DATA_BLOCK "RSE_GLOBAL_DB"
TITLE = Report System Error Diagnostic Block
{ S7_Optimized_Access := 'FALSE' }
AUTHOR : SIMATIC
FAMILY : RSEDIAG
NAME : RSE
VERSION : 1.0
NON_RETAIN
// This DB contains the generated data from STEP 7 Report System Errors.
   STRUCT
      DB_Nummer { ExternalVisible := 'False'} : Word;
      DB_Init { ExternalVisible := 'False'} : Bool;
      HotRestart { ExternalVisible := 'False'} : Bool;
      DB_bZaehler { ExternalVisible := 'False'} : Byte;
      TraceZyklusNo { ExternalVisible := 'False'} : Word;
      TraceZyklusAuswertung { ExternalVisible := 'False'} : Word;
      TraceZyklus126No { ExternalVisible := 'False'} : Word;
      TraceZyklus127No { ExternalVisible := 'False'} : Word;
      TraceStatus1 { ExternalVisible := 'False'} : Word;
      TraceMeldungenAnzahl { ExternalVisible := 'False'} : Byte;
      TraceMeldungenMax { ExternalVisible := 'False'} : Byte;
      Daten { ExternalVisible := 'False'} : Array[1..805] of Byte;
      DiagSZLHeader { ExternalVisible := 'False'} : Struct
         LENTHDR { ExternalVisible := 'False'} : Word;
         N_DR { ExternalVisible := 'False'} : Word;
      END_STRUCT;
      SZLHeader { ExternalVisible := 'False'} : Struct
         LENTHDR { ExternalVisible := 'False'} : Word;
         N_DR { ExternalVisible := 'False'} : Word;
      END_STRUCT;
   END_STRUCT;


BEGIN
   DB_Nummer := WORD#16#0032;
   Daten[1] := BYTE#16#08;
   Daten[4] := BYTE#16#09;
   Daten[5] := BYTE#16#03;
   Daten[6] := BYTE#16#58;
   Daten[7] := BYTE#16#03;
   Daten[8] := BYTE#16#26;
   Daten[9] := BYTE#16#03;
   Daten[10] := BYTE#16#28;
   Daten[11] := BYTE#16#03;
   Daten[12] := BYTE#16#2A;
   Daten[13] := BYTE#16#03;
   Daten[14] := BYTE#16#2C;
   Daten[15] := BYTE#16#03;
   Daten[16] := BYTE#16#2E;
   Daten[17] := BYTE#16#03;
   Daten[18] := BYTE#16#30;
   Daten[19] := BYTE#16#03;
   Daten[20] := BYTE#16#56;
   Daten[21] := BYTE#16#03;
   Daten[22] := BYTE#16#3C;
   Daten[23] := BYTE#16#01;
   Daten[29] := BYTE#16#08;
   Daten[30] := BYTE#16#40;
   Daten[32] := BYTE#16#04;
   Daten[33] := BYTE#16#03;
   Daten[34] := BYTE#16#66;
   Daten[35] := BYTE#16#03;
   Daten[36] := BYTE#16#46;
   Daten[37] := BYTE#16#03;
   Daten[38] := BYTE#16#44;
   Daten[39] := BYTE#16#03;
   Daten[40] := BYTE#16#42;
   Daten[51] := BYTE#16#FF;
   Daten[52] := BYTE#16#FF;
   Daten[53] := BYTE#16#FF;
   Daten[54] := BYTE#16#FF;
   Daten[56] := BYTE#16#40;
   Daten[67] := BYTE#16#FF;
   Daten[68] := BYTE#16#FF;
   Daten[69] := BYTE#16#FF;
   Daten[70] := BYTE#16#FF;
   Daten[71] := BYTE#16#03;
   Daten[72] := BYTE#16#48;
   Daten[75] := BYTE#16#04;
   Daten[79] := BYTE#16#08;
   Daten[80] := BYTE#16#08;
   Daten[85] := BYTE#16#FF;
   Daten[86] := BYTE#16#FF;
   Daten[87] := BYTE#16#FF;
   Daten[88] := BYTE#16#FF;
   Daten[93] := BYTE#16#05;
   Daten[95] := BYTE#16#06;
   Daten[99] := BYTE#16#20;
   Daten[100] := BYTE#16#04;
   Daten[109] := BYTE#16#01;
   Daten[110] := BYTE#16#FF;
   Daten[111] := BYTE#16#FF;
   Daten[112] := BYTE#16#FF;
   Daten[113] := BYTE#16#FF;
   Daten[114] := BYTE#16#07;
   Daten[116] := BYTE#16#08;
   Daten[118] := BYTE#16#05;
   Daten[120] := BYTE#16#06;
   Daten[123] := BYTE#16#20;
   Daten[124] := BYTE#16#04;
   Daten[133] := BYTE#16#01;
   Daten[134] := BYTE#16#FF;
   Daten[135] := BYTE#16#FF;
   Daten[136] := BYTE#16#FF;
   Daten[137] := BYTE#16#FF;
   Daten[138] := BYTE#16#07;
   Daten[140] := BYTE#16#08;
   Daten[142] := BYTE#16#05;
   Daten[144] := BYTE#16#06;
   Daten[147] := BYTE#16#20;
   Daten[148] := BYTE#16#04;
   Daten[152] := BYTE#16#08;
   Daten[153] := BYTE#16#08;
   Daten[157] := BYTE#16#FF;
   Daten[158] := BYTE#16#FF;
   Daten[159] := BYTE#16#FF;
   Daten[160] := BYTE#16#FF;
   Daten[161] := BYTE#16#FF;
   Daten[162] := BYTE#16#09;
   Daten[166] := BYTE#16#08;
   Daten[168] := BYTE#16#20;
   Daten[169] := BYTE#16#04;
   Daten[173] := BYTE#16#08;
   Daten[174] := BYTE#16#08;
   Daten[178] := BYTE#16#FF;
   Daten[179] := BYTE#16#FF;
   Daten[180] := BYTE#16#FF;
   Daten[181] := BYTE#16#FF;
   Daten[182] := BYTE#16#FF;
   Daten[183] := BYTE#16#09;
   Daten[187] := BYTE#16#08;
   Daten[189] := BYTE#16#20;
   Daten[190] := BYTE#16#04;
   Daten[194] := BYTE#16#08;
   Daten[195] := BYTE#16#08;
   Daten[199] := BYTE#16#FF;
   Daten[200] := BYTE#16#FF;
   Daten[201] := BYTE#16#FF;
   Daten[202] := BYTE#16#FF;
   Daten[203] := BYTE#16#FF;
   Daten[204] := BYTE#16#09;
   Daten[208] := BYTE#16#08;
   Daten[210] := BYTE#16#20;
   Daten[211] := BYTE#16#04;
   Daten[215] := BYTE#16#08;
   Daten[216] := BYTE#16#08;
   Daten[220] := BYTE#16#FF;
   Daten[221] := BYTE#16#FF;
   Daten[222] := BYTE#16#FF;
   Daten[223] := BYTE#16#FF;
   Daten[224] := BYTE#16#FF;
   Daten[225] := BYTE#16#09;
   Daten[229] := BYTE#16#08;
   Daten[231] := BYTE#16#20;
   Daten[232] := BYTE#16#04;
   Daten[236] := BYTE#16#08;
   Daten[237] := BYTE#16#08;
   Daten[241] := BYTE#16#FF;
   Daten[242] := BYTE#16#FF;
   Daten[243] := BYTE#16#FF;
   Daten[244] := BYTE#16#FF;
   Daten[245] := BYTE#16#FF;
   Daten[246] := BYTE#16#09;
   Daten[250] := BYTE#16#08;
   Daten[253] := BYTE#16#04;
   Daten[257] := BYTE#16#08;
   Daten[258] := BYTE#16#08;
   Daten[263] := BYTE#16#FF;
   Daten[264] := BYTE#16#FF;
   Daten[265] := BYTE#16#FF;
   Daten[266] := BYTE#16#FF;
   Daten[273] := BYTE#16#40;
   Daten[284] := BYTE#16#FF;
   Daten[285] := BYTE#16#FF;
   Daten[286] := BYTE#16#FF;
   Daten[287] := BYTE#16#FF;
   Daten[288] := BYTE#16#03;
   Daten[289] := BYTE#16#5C;
   Daten[292] := BYTE#16#04;
   Daten[296] := BYTE#16#08;
   Daten[297] := BYTE#16#08;
   Daten[302] := BYTE#16#FF;
   Daten[303] := BYTE#16#FF;
   Daten[304] := BYTE#16#FF;
   Daten[305] := BYTE#16#FF;
   Daten[311] := BYTE#16#08;
   Daten[312] := BYTE#16#48;
   Daten[314] := BYTE#16#04;
   Daten[315] := BYTE#16#03;
   Daten[316] := BYTE#16#3E;
   Daten[317] := BYTE#16#03;
   Daten[318] := BYTE#16#18;
   Daten[319] := BYTE#16#03;
   Daten[320] := BYTE#16#1A;
   Daten[321] := BYTE#16#03;
   Daten[322] := BYTE#16#4A;
   Daten[323] := BYTE#16#01;
   Daten[329] := BYTE#16#02;
   Daten[332] := BYTE#16#40;
   Daten[343] := BYTE#16#FF;
   Daten[344] := BYTE#16#FF;
   Daten[345] := BYTE#16#FF;
   Daten[346] := BYTE#16#FF;
   Daten[348] := BYTE#16#20;
   Daten[349] := BYTE#16#04;
   Daten[353] := BYTE#16#08;
   Daten[354] := BYTE#16#08;
   Daten[355] := BYTE#16#FF;
   Daten[356] := BYTE#16#FF;
   Daten[357] := BYTE#16#FF;
   Daten[358] := BYTE#16#FF;
   Daten[359] := BYTE#16#FF;
   Daten[360] := BYTE#16#FF;
   Daten[361] := BYTE#16#FF;
   Daten[362] := BYTE#16#FF;
   Daten[363] := BYTE#16#09;
   Daten[367] := BYTE#16#20;
   Daten[369] := BYTE#16#20;
   Daten[370] := BYTE#16#04;
   Daten[374] := BYTE#16#08;
   Daten[375] := BYTE#16#08;
   Daten[376] := BYTE#16#FF;
   Daten[377] := BYTE#16#FF;
   Daten[378] := BYTE#16#FF;
   Daten[379] := BYTE#16#FF;
   Daten[380] := BYTE#16#FF;
   Daten[381] := BYTE#16#FF;
   Daten[382] := BYTE#16#FF;
   Daten[383] := BYTE#16#FF;
   Daten[384] := BYTE#16#09;
   Daten[388] := BYTE#16#20;
   Daten[390] := BYTE#16#20;
   Daten[391] := BYTE#16#04;
   Daten[395] := BYTE#16#08;
   Daten[396] := BYTE#16#08;
   Daten[400] := BYTE#16#FF;
   Daten[401] := BYTE#16#FF;
   Daten[402] := BYTE#16#FF;
   Daten[403] := BYTE#16#FF;
   Daten[404] := BYTE#16#FF;
   Daten[405] := BYTE#16#09;
   Daten[409] := BYTE#16#08;
   Daten[410] := BYTE#16#08;
   Daten[411] := BYTE#16#48;
   Daten[413] := BYTE#16#03;
   Daten[414] := BYTE#16#03;
   Daten[415] := BYTE#16#64;
   Daten[416] := BYTE#16#03;
   Daten[417] := BYTE#16#22;
   Daten[418] := BYTE#16#03;
   Daten[419] := BYTE#16#54;
   Daten[420] := BYTE#16#01;
   Daten[426] := BYTE#16#02;
   Daten[429] := BYTE#16#40;
   Daten[440] := BYTE#16#FF;
   Daten[441] := BYTE#16#FF;
   Daten[442] := BYTE#16#FF;
   Daten[443] := BYTE#16#FF;
   Daten[446] := BYTE#16#04;
   Daten[450] := BYTE#16#08;
   Daten[451] := BYTE#16#08;
   Daten[456] := BYTE#16#FF;
   Daten[457] := BYTE#16#FF;
   Daten[458] := BYTE#16#FF;
   Daten[459] := BYTE#16#FF;
   Daten[460] := BYTE#16#09;
   Daten[465] := BYTE#16#04;
   Daten[469] := BYTE#16#08;
   Daten[470] := BYTE#16#08;
   Daten[475] := BYTE#16#FF;
   Daten[476] := BYTE#16#FF;
   Daten[477] := BYTE#16#FF;
   Daten[478] := BYTE#16#FF;
   Daten[479] := BYTE#16#09;
   Daten[482] := BYTE#16#08;
   Daten[483] := BYTE#16#48;
   Daten[485] := BYTE#16#03;
   Daten[486] := BYTE#16#03;
   Daten[487] := BYTE#16#62;
   Daten[488] := BYTE#16#03;
   Daten[489] := BYTE#16#1C;
   Daten[490] := BYTE#16#03;
   Daten[491] := BYTE#16#4C;
   Daten[492] := BYTE#16#01;
   Daten[498] := BYTE#16#02;
   Daten[501] := BYTE#16#40;
   Daten[512] := BYTE#16#FF;
   Daten[513] := BYTE#16#FF;
   Daten[514] := BYTE#16#FF;
   Daten[515] := BYTE#16#FF;
   Daten[518] := BYTE#16#04;
   Daten[522] := BYTE#16#08;
   Daten[523] := BYTE#16#08;
   Daten[528] := BYTE#16#FF;
   Daten[529] := BYTE#16#FF;
   Daten[530] := BYTE#16#FF;
   Daten[531] := BYTE#16#FF;
   Daten[532] := BYTE#16#09;
   Daten[537] := BYTE#16#04;
   Daten[541] := BYTE#16#08;
   Daten[542] := BYTE#16#08;
   Daten[547] := BYTE#16#FF;
   Daten[548] := BYTE#16#FF;
   Daten[549] := BYTE#16#FF;
   Daten[550] := BYTE#16#FF;
   Daten[551] := BYTE#16#09;
   Daten[554] := BYTE#16#08;
   Daten[555] := BYTE#16#48;
   Daten[557] := BYTE#16#03;
   Daten[558] := BYTE#16#03;
   Daten[559] := BYTE#16#5E;
   Daten[560] := BYTE#16#03;
   Daten[561] := BYTE#16#1E;
   Daten[562] := BYTE#16#03;
   Daten[563] := BYTE#16#4E;
   Daten[564] := BYTE#16#01;
   Daten[570] := BYTE#16#02;
   Daten[573] := BYTE#16#40;
   Daten[584] := BYTE#16#FF;
   Daten[585] := BYTE#16#FF;
   Daten[586] := BYTE#16#FF;
   Daten[587] := BYTE#16#FF;
   Daten[590] := BYTE#16#04;
   Daten[594] := BYTE#16#08;
   Daten[595] := BYTE#16#08;
   Daten[600] := BYTE#16#FF;
   Daten[601] := BYTE#16#FF;
   Daten[602] := BYTE#16#FF;
   Daten[603] := BYTE#16#FF;
   Daten[604] := BYTE#16#09;
   Daten[609] := BYTE#16#04;
   Daten[613] := BYTE#16#08;
   Daten[614] := BYTE#16#08;
   Daten[619] := BYTE#16#FF;
   Daten[620] := BYTE#16#FF;
   Daten[621] := BYTE#16#FF;
   Daten[622] := BYTE#16#FF;
   Daten[623] := BYTE#16#09;
   Daten[626] := BYTE#16#08;
   Daten[627] := BYTE#16#48;
   Daten[629] := BYTE#16#03;
   Daten[630] := BYTE#16#03;
   Daten[631] := BYTE#16#60;
   Daten[632] := BYTE#16#03;
   Daten[633] := BYTE#16#20;
   Daten[634] := BYTE#16#03;
   Daten[635] := BYTE#16#52;
   Daten[636] := BYTE#16#01;
   Daten[642] := BYTE#16#02;
   Daten[645] := BYTE#16#40;
   Daten[656] := BYTE#16#FF;
   Daten[657] := BYTE#16#FF;
   Daten[658] := BYTE#16#FF;
   Daten[659] := BYTE#16#FF;
   Daten[662] := BYTE#16#04;
   Daten[666] := BYTE#16#08;
   Daten[667] := BYTE#16#08;
   Daten[672] := BYTE#16#FF;
   Daten[673] := BYTE#16#FF;
   Daten[674] := BYTE#16#FF;
   Daten[675] := BYTE#16#FF;
   Daten[676] := BYTE#16#09;
   Daten[681] := BYTE#16#04;
   Daten[685] := BYTE#16#08;
   Daten[686] := BYTE#16#08;
   Daten[691] := BYTE#16#FF;
   Daten[692] := BYTE#16#FF;
   Daten[693] := BYTE#16#FF;
   Daten[694] := BYTE#16#FF;
   Daten[695] := BYTE#16#09;
   Daten[698] := BYTE#16#08;
   Daten[699] := BYTE#16#48;
   Daten[701] := BYTE#16#03;
   Daten[702] := BYTE#16#03;
   Daten[703] := BYTE#16#5A;
   Daten[704] := BYTE#16#03;
   Daten[705] := BYTE#16#24;
   Daten[706] := BYTE#16#03;
   Daten[707] := BYTE#16#50;
   Daten[708] := BYTE#16#01;
   Daten[714] := BYTE#16#02;
   Daten[717] := BYTE#16#40;
   Daten[728] := BYTE#16#FF;
   Daten[729] := BYTE#16#FF;
   Daten[730] := BYTE#16#FF;
   Daten[731] := BYTE#16#FF;
   Daten[734] := BYTE#16#04;
   Daten[738] := BYTE#16#08;
   Daten[739] := BYTE#16#08;
   Daten[744] := BYTE#16#FF;
   Daten[745] := BYTE#16#FF;
   Daten[746] := BYTE#16#FF;
   Daten[747] := BYTE#16#FF;
   Daten[748] := BYTE#16#09;
   Daten[753] := BYTE#16#04;
   Daten[757] := BYTE#16#08;
   Daten[758] := BYTE#16#08;
   Daten[763] := BYTE#16#FF;
   Daten[764] := BYTE#16#FF;
   Daten[765] := BYTE#16#FF;
   Daten[766] := BYTE#16#FF;
   Daten[767] := BYTE#16#09;
   Daten[770] := BYTE#16#08;
   Daten[771] := BYTE#16#08;
   Daten[773] := BYTE#16#06;
   Daten[774] := BYTE#16#03;
   Daten[775] := BYTE#16#40;
   Daten[776] := BYTE#16#03;
   Daten[777] := BYTE#16#34;
   Daten[778] := BYTE#16#03;
   Daten[779] := BYTE#16#36;
   Daten[780] := BYTE#16#03;
   Daten[781] := BYTE#16#38;
   Daten[782] := BYTE#16#03;
   Daten[783] := BYTE#16#32;
   Daten[784] := BYTE#16#03;
   Daten[785] := BYTE#16#3A;
   Daten[786] := BYTE#16#03;
   Daten[792] := BYTE#16#03;
   Daten[793] := BYTE#16#66;
   Daten[794] := BYTE#16#01;
   Daten[803] := BYTE#16#03;
   Daten[804] := BYTE#16#56;
   Daten[805] := BYTE#16#B4;

END_DATA_BLOCK

